(*			
	RafalOS
	Rafał Osajda		20.11.2025		TC 4024.66
	Interfejs umożliwający wywoływanie moted z HMIManager
*)
INTERFACE ITF_MCHMIMachineControl_HMI EXTENDS ITF_BaseTopElement_HMI

METHOD PUBLIC AddPrepareScreenModuleFromManager : BOOL
VAR_INPUT
	itfModule	: ITF_MCHMIPrepareScreen_Init;// ITF_MCHMIPrepareDataForScreen;
END_VAR
END_METHOD

(*			
	RafalOS
	Rafał Osajda		19.11.2025		TC 4024.66
	Sprzątanie po stronie wywoływane z HMIManager i wywołująca odpowiednią metode z ITF z arrPrepareScreen
*)
METHOD ClearAfterScreenFroHMIManager : BOOL
VAR_INPUT
	iScreen		: INT;
	iMode		: INT;
END_VAR
END_METHOD

METHOD PUBLIC LinkMachineControlData : BOOL
VAR_INPUT
	stData			: REFERENCE TO ST_MCHMIMachineControl_HMI_Link;
END_VAR
END_METHOD

(*			
	RafalOS
	Rafał Osajda		20.11.2025		TC 4024.66
	Podpięcie modułu generowania danych do odpowiedniej pozycji w tablicy [Okno][Tryb]
*)
METHOD PUBLIC LinkPrepareScreenToArrayFromConfiguration : BOOL
VAR_INPUT
	iScreen		: INT;
	iMode		: INT;
	itfModule	: ITF_MCHMIPrepareDataForScreen;
END_VAR
END_METHOD

(*			
	RafalOS
	Rafał Osajda		19.11.2025		TC 4024.66
	Przygotowanie danych dla strony wywoływane z HMIManager i wywołująca odpowiednią metode z ITF z arrPrepareScreen
*)
METHOD PrepareDataForScreenFromHMIManager : BOOL
VAR_INPUT
	iScreen		: INT;
	iMode		: INT;
END_VAR
END_METHOD

(*			
	RafalOS
	Rafał Osajda		19.11.2025		TC 4024.66
	Przygotowanie strony wywoływane z HMIManager i wywołująca odpowiednią metode z ITF z arrPrepareScreen
*)
METHOD PrepareForScreenFromHMIManager : BOOL
VAR_INPUT
	iScreen		: INT;
	iMode		: INT;
END_VAR
END_METHOD

END_INTERFACE

(* stored: Version 1.1.0.1
   Itf ITF_MCHMIMachineControl_HMI: Id {6538430b-c357-0110-090b-55567298ce9d}
   Method AddPrepareScreenModuleFromManager: Id {aca03413-ab44-0db0-2798-45d6c1e55008}
   Method ClearAfterScreenFroHMIManager: Id {f45baa25-757c-0fe6-219c-a44fc4762619}
   Method LinkMachineControlData: Id {5b1d074d-68af-002e-0084-5fe1502c4b5b}
   Method LinkPrepareScreenToArrayFromConfiguration: Id {6019ac61-4b85-0056-06ad-6c9ca798e7f8}
   Method PrepareDataForScreenFromHMIManager: Id {19732316-0985-0bc4-10a0-bbeee6760cf3}
   Method PrepareForScreenFromHMIManager: Id {ab08d887-ef68-0904-2cb0-dfdd188c94ac} *)
